PROGRAM MAIN
VAR
	sad: DINT;
END_VAR

sad := 1 +sad;

END_PROGRAM

(* stored: Version 1.1.0.1, ProductVersion 3.1.4024.10
   POU MAIN: Id {3f11ceaa-009a-4b5e-9a63-7b2c8a282994}, SpecialFunc None *)
